Universal Robots PolyScope program: Hospital_base.urp

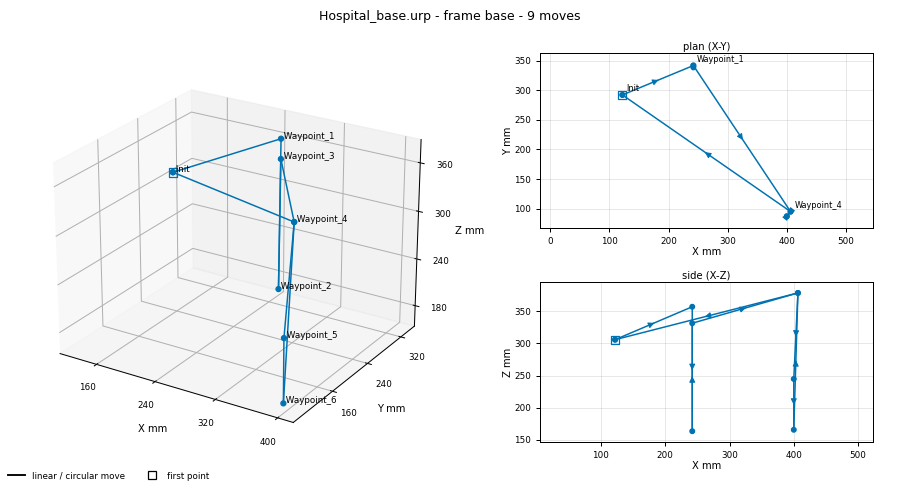
[picture p0: tool path of Hospital_base.urp in frame base, 9 of 9 moves have a stored position in this frame; points joined in program order, loops and branches not executed]
Program Hospital_base (installation=default directory=/programs/Mursal createdIn=5.11.11.1010533 lastSavedIn=5.11.11.1010533 robotSerialNumber=20205300864)
Calibrated DH parameters: a=[-0.000166, -0.243494, -0.153108, 0.000057, -0.000123, 0]; d=[0.151897, -1.34267, 53.988124, -52.514559, 0.085283, 0.092193]; alpha=[1.572472, -0.003756, 0.002824, 1.570807, -1.572621, 0]; deltaTheta=[0, 0.020704, 7.033215, -0.770746, 0.000004, 0]
Robot Program (runOnlyOnce=true)
  MoveL speed 250 mm/s, acceleration 1200 mm/s^2 (useActiveTCP=true) feature=Base
    Waypoint Init: TCP in base x=122.112 y=292.107 z=305.722 mm, rx=1.1347 ry=-2.9295 rz=0.0001 rad; joints [91.642, -87.585, -91.768, -90.546, 90.033, 859.396] deg
    Waypoint Waypoint_1: TCP in base x=242.037 y=341.762 z=356.872 mm, rx=2.253 ry=-2.1894 rz=0 rad; joints [72.907, -118.45, -38.628, -112.818, 89.869, 791.31] deg
    Waypoint Waypoint_2: TCP in base x=242.067 y=338.572 z=163.434 mm, rx=-2.2529 ry=2.1894 rz=-0.0001 rad; joints [72.656, -120.738, -88.952, -60.202, 89.949, 791.167] deg
    URCap Gripper (Robotiq_Grippers, Robotiq Inc.) dataModel(position=100.0, force=12.0, speed=100.0, positionInDouble=100.0, forceInDouble=12.0, speedInDouble=100.0, slaveIds=[9], blocking=true, robotCompliant=false)
    Waypoint Waypoint_3: TCP in base x=242.024 y=341.771 z=331.286 mm, rx=-2.253 ry=2.1894 rz=0.0001 rad; joints [72.883, -115.712, -50.14, -104.041, 89.902, 791.302] deg
    Waypoint Waypoint_4: TCP in base x=406.298 y=94.923 z=378.345 mm, rx=3.141 ry=0.0607 rz=-0.0001 rad; joints [31.463, -122.167, -25.973, -121.757, 89.833, 659.277] deg
    Waypoint Waypoint_5: TCP in base x=399.867 y=86.92 z=244.634 mm, rx=-3.1155 ry=0.0042 rz=-0.0713 rad; joints [30.858, -111.545, -80.987, -74.372, 89.853, 1021.124] deg
    Waypoint Waypoint_6: TCP in base x=399.874 y=86.963 z=165.636 mm, rx=-3.1152 ry=0.004 rz=-0.0721 rad; joints [30.833, -118.573, -93.306, -54.986, 89.851, 1021.132] deg
    URCap Gripper (Robotiq_Grippers, Robotiq Inc.) dataModel(position=0.0, force=0.0, speed=100.0, positionInDouble=0.0, forceInDouble=0.0, speedInDouble=100.0, slaveIds=[9], blocking=true, robotCompliant=false)
    Waypoint Waypoint_4: TCP in base x=406.298 y=94.923 z=378.345 mm, rx=3.141 ry=0.0607 rz=-0.0001 rad; joints [31.463, -122.167, -25.973, -121.757, 89.833, 659.277] deg
    Waypoint Init: TCP in base x=122.112 y=292.107 z=305.722 mm, rx=1.1347 ry=-2.9295 rz=0.0001 rad; joints [91.642, -87.585, -91.768, -90.546, 90.033, 859.396] deg
